(* CoDeSys 2.3 library: Lib_MQTT_Publisher_01.lib *)
(* Libraries: Lib_DebugLogger_01.lib 18.7.17 20:48:14, C:\Program Files (x86)\WAGO Software\CoDeSys V2.3\Targets\WAGO\Libraries\32_Bit\SysLibSockets.lib 10.2.11 09:20:54, C:\Program Files (x86)\WAGO Software\CoDeSys V2.3\Targets\WAGO\Libraries\Application\WagoLibEthernet_01.lib 1.4.15 14:24:28, Standard.lib 2.6.14 10:37:46, Util.lib 26.9.14 10:12:46 *)

(* Data type *)
TYPE Buffer :
STRUCT
	data : ARRAY [0..MAX_RECEIVE_TCP_CLIENT] OF BYTE;
	iPos : DWORD := 0;
END_STRUCT
END_TYPE

(* Data type *)
TYPE ConnectFlags :
STRUCT
	xUsername     : BOOL;
	xPassword     : BOOL;
	xWillRetain   : BOOL;
	xWillQoS1     : BOOL;
    xWillQoS2     : BOOL;
	xWillFlag     : BOOL;
	xCleanSession : BOOL;
END_STRUCT
END_TYPE

(* Data type *)
TYPE E_MQTT_MAIN_STATE : (

	eMQTT_NO_TCP_CONNECTION,
	eMQTT_CONNECTED,
	eMQTT_NOT_CONNECTED,
	eMQTT_TIMEOUT,
	eMQTT_WAIT_RESPONSE
);
END_TYPE

(* Data type *)
TYPE FixedHeader :
STRUCT
	bMessageType : BYTE := 16#00;
	xDUP_FLAG    : BOOL := FALSE;
	xQos         : BYTE := 16#00; (*0,1,2*)
	xRetain      : BOOL := FALSE;
END_STRUCT
END_TYPE

(* Data type *)
TYPE stMQTT_Config :
STRUCT
	sIdentifier : STRING := 'wagoPLC';
	sIp : STRING;
	wPortNumber : WORD := 1883;
	sUsername : STRING;
	sPassword : STRING;
END_STRUCT
END_TYPE

(* POU _BUFFER_CONCAT, ST *)
FUNCTION _BUFFER_CONCAT : BOOL
VAR_INPUT
	PT  : POINTER TO Buffer;
	PTContact  : POINTER TO Buffer;
END_VAR
VAR
	i: INT;
END_VAR
FOR i:=0 TO DWORD_TO_INT(PTContact^.iPos) -1 BY 1 DO
	_BUFFER_PUSH(PT, PTContact^.data[i]);
END_FOR
END_FUNCTION

(* POU _BUFFER_PUSH, ST *)
FUNCTION _BUFFER_PUSH : BOOL
VAR_INPUT
	PT  : POINTER TO Buffer;
	IN  : BYTE;
END_VAR

VAR
END_VAR
(* pushed data to a buffer array *)
PT^.data[PT^.iPos] := IN;

PT^.iPos := PT^.iPos + 1;

_BUFFER_PUSH := TRUE;
END_FUNCTION

(* POU _BUFFER_PUSH_STRING, ST *)
FUNCTION _BUFFER_PUSH_STRING : BOOL
VAR_INPUT
	PT : POINTER TO Buffer;
	IN : STRING(255);
	INCLUDE_LENGTH : BOOL := FALSE;
END_VAR
VAR
	sPT : POINTER TO BYTE;
	iLen : DWORD;
	i : DWORD;
	nxtPtr: POINTER TO BYTE;
END_VAR
iLen := LEN(IN);
sPT := ADR(IN);

IF INCLUDE_LENGTH THEN

(*
	_BUFFER_PUSH(PT, BYTE_OF_DWORD(iLen,1));
	_BUFFER_PUSH(PT, BYTE_OF_DWORD(iLen,0));
*)

		_BUFFER_PUSH(PT, DWORD_TO_BYTE(SHR(iLen,8)));
		_BUFFER_PUSH(PT, DWORD_TO_BYTE(iLen));

END_IF

FOR i:=0 TO iLen-1 BY 1 DO
	nxtPtr := sPT + i * SIZEOF(sPT^);
	_BUFFER_PUSH(PT, nxtPtr^);
END_FOR
END_FUNCTION

(* POU _BUFFER_SET, ST *)
FUNCTION _BUFFER_SET : BOOL
VAR_INPUT
	PT  : POINTER TO Buffer;
	IN  : BYTE;
	POS : UINT := 0;
END_VAR
VAR
END_VAR
PT^.data[POS] := IN;

IF PT^.iPos < POS THEN
	PT^.iPos := POS;
END_IF
END_FUNCTION

(* POU CREATE_MESSAGE, ST *)
FUNCTION CREATE_MESSAGE : BOOL
VAR_INPUT
	PT          : POINTER TO Buffer;
	fixedHeader     : FixedHeader;
	variableHeader  : Buffer;
	payLoad         : Buffer;
END_VAR
VAR
	bTemp  : BYTE;
	remainingLength: DWORD;
END_VAR
(* FIXED HEADER *)
(* BYTE 1 *)
bTemp := bTemp OR SHL(fixedHeader.bMessageType, 4) OR SHL(FixedHeader.xQos, 1);

bTemp.3 := FixedHeader.xDUP_FLAG;
bTemp.0 := FixedHeader.xRetain;

_BUFFER_PUSH(PT, bTemp);

(* BYTE 2 *)
remainingLength := variableHeader.iPos + payLoad.iPos;

ENCODE_REMAINING_LENGTH(PT, remainingLength);
(*_BUFFER_PUSH(PT, remainingLength);*)

(* VARIABLE HEADER *)
_BUFFER_CONCAT(PT, ADR(variableHeader));

(* PAYLOAD *)
_BUFFER_CONCAT(PT, ADR(payLoad));
END_FUNCTION

(* POU ENCODE_REMAINING_LENGTH, ST *)
FUNCTION ENCODE_REMAINING_LENGTH : BOOL
VAR_INPUT
	PT : POINTER TO Buffer;
	LENGTH : DWORD;
END_VAR
VAR
	wPt : POINTER TO DWORD; (*4 bytes*)
	digit: DWORD;
END_VAR
wPt := ADR(LENGTH);

IF LENGTH = 0 THEN
	_BUFFER_PUSH(PT, 16#00);
	RETURN;
END_IF

WHILE LENGTH > 0 DO
	digit := LENGTH MOD 128;
	LENGTH := LENGTH / 128;
	
	IF LENGTH > 0 THEN
		digit := digit OR 16#80;
	END_IF
(*	_BUFFER_PUSH(PT, BYTE_OF_DWORD(digit,0));*)
	_BUFFER_PUSH(PT, DWORD_TO_BYTE(digit));
END_WHILE
END_FUNCTION

(* POU MQTT_Client, ST *)
FUNCTION_BLOCK MQTT_Client

VAR_INPUT
	sTopic: STRING;
	sPayload: STRING(255);
	sIp : STRING;
	iPortNumber : WORD;
	sUsername : STRING;
	sPassword : STRING;
END_VAR

VAR_IN_OUT
	xPublish: BOOL;
END_VAR

VAR_OUTPUT
	xConnected : BOOL := FALSE;
	xBusy : BOOL := FALSE;
END_VAR

VAR
	sendBuffer : 				Buffer;
	receiveBuffer :				Buffer;

	fixedHeader: 				FixedHeader;
	variableHeader: 			Buffer;

	payLoad:  					Buffer;

	connectFlags: 			ConnectFlags;
	tcpClient: 					TCP_Client;
	xStartSend 					: BOOL 					:= FALSE;
	diReceiveCount 				: DINT;
	connectionTimer				: TON;
	xTimeOut 					: BOOL;
	iIncomingMessageType		: BYTE;
	eState						: E_MQTT_MAIN_STATE 	:= eMQTT_NO_TCP_CONNECTION;
	xStartTimer					: BOOL;


	xOpenConnection: BOOL;



	bEntry: BOOL := TRUE;
	DebugLog: BOOL;
END_VAR

VAR CONSTANT
	CONNECTION_TIMEOUT : TIME := t#10s;


	Reserved   	: BYTE := 0;
	CONNECT     : BYTE := 1;
	CONNACK     : BYTE := 2;
	PUBLISH     : BYTE := 3;
	PUBACK      : BYTE := 4;
	PUBREC      : BYTE := 5;
	PUBREL      : BYTE := 6;
	PUBCOMP     : BYTE := 7;
	SUBSCRIBE   : BYTE := 8;
	SUBACK      : BYTE := 9;
	UNSUBSCRIBE : BYTE := 10;
	UNSUBACK    : BYTE := 11;
	PINGREQ     : BYTE := 12;
	PINGRESP    : BYTE := 13;
	DISCONNECT  : BYTE := 14;
	Reserved2   : BYTE := 15;

END_VAR
tcpClient(
	xOpenConnection		:= xOpenConnection,
	sIPaddress			:= sIp ,
	wPortNumber			:= iPortNumber,
	ptSendData 			:= ADR(sendBuffer.data),
	diSendCount 			:= sendBuffer.iPos,
	xStartSend 			:= xStartSend,
	aReceiveBuffer		:= receiveBuffer.data,
	diReceiveCount		:= diReceiveCount ,
	xConnected=> ,
	diError=> );

connectionTimer(
	IN:=xStartTimer,
	PT:=CONNECTION_TIMEOUT-t#2s,
	Q => xTimeOut);

(* INIT *)
payLoad.iPos := 0;
variableHeader.iPos := 0;

IF xTimeOut THEN
	eState := eMQTT_TIMEOUT;
END_IF

(* Execute current state *)

(*Global TCP Connection Check*)

IF 		(NOT tcpClient.xConnected OR tcpClient.diError <> 0)
	AND eState <> eMQTT_NO_TCP_CONNECTION THEN
	DebugLog('connection lost', INFO);
	DebugLog(DINT_TO_STRING(tcpClient.diError), INFO);
	eState := eMQTT_NO_TCP_CONNECTION;
	bEntry := TRUE;
END_IF;



CASE eState OF


	eMQTT_NO_TCP_CONNECTION:
		IF bEntry THEN
			bEntry := FALSE;
			xOpenConnection := FALSE;
			xStartSend := FALSE;
			xConnected := FALSE;
			DebugLog('try to connect', INFO);

		ELSE
			xOpenConnection := TRUE;
			IF tcpClient.xConnected THEN
				eState := eMQTT_NOT_CONNECTED;
				bEntry := TRUE;
			END_IF

		END_IF




	eMQTT_CONNECTED:
			IF diReceiveCount > 0 THEN
				iIncomingMessageType := receiveBuffer.data[0];
				IF iIncomingMessageType = SHL(PINGRESP, 4) THEN
					xStartTimer := TRUE;
				END_IF
				diReceiveCount := 0;
			END_IF
	
			IF xPublish THEN
				fixedHeader.bMessageType := PUBLISH;
				fixedHeader.xDUP_FLAG := FALSE;
				fixedHeader.xQos := 16#00; (* only QoS 0 supported *)
				fixedHeader.xRetain := FALSE;
		
				_BUFFER_PUSH_STRING(ADR(variableHeader), sTopic, TRUE); (* Topic *)
				IF fixedHeader.xQos > 16#00 THEN
					_BUFFER_PUSH(ADR(variableHeader), 16#00);(* Message ID *)
					_BUFFER_PUSH(ADR(variableHeader), 16#00);
				END_IF
	
				_BUFFER_PUSH_STRING(ADR(payLoad), sPayload, FALSE);
		
				sendBuffer.iPos := 0;
				CREATE_MESSAGE(ADR(sendBuffer), fixedHeader, variableHeader, payLoad);
	
				xStartSend := TRUE;
		
				xPublish := FALSE;

			END_IF



	eMQTT_NOT_CONNECTED:

			sendBuffer.iPos := 0;
			xStartTimer := FALSE;
			fixedHeader.bMessageType := CONNECT;
	
			_BUFFER_PUSH_STRING(
				ADR(variableHeader),
				'MQIsdp',
				TRUE); (* Protocol Name*)
			_BUFFER_PUSH(
				ADR(variableHeader),
				 3); (* Version Number*)
	
			connectFlags.xCleanSession 	:= TRUE;
			connectFlags.xWillFlag     		:= FALSE;
			connectFlags.xWillQoS1    	 	:= FALSE;
			connectFlags.xWillQoS2     		:= FALSE;
			connectFlags.xWillRetain   		:= FALSE;
			connectFlags.xUsername 		:= LEN(sUsername) > 0;
			connectFlags.xPassword 		:= LEN(sPassword) > 0;
	
			_BUFFER_PUSH(
				ADR(variableHeader),
				 PACK(		FALSE,
							connectFlags.xCleanSession,
							connectFlags.xWillFlag,
							connectFlags.xWillQoS1,
							connectFlags.xWillQoS2,
							connectFlags.xWillRetain,
							connectFlags.xPassword,
							connectFlags.xUsername));
	
			_BUFFER_PUSH(ADR(variableHeader), 16#00);
			_BUFFER_PUSH(ADR(variableHeader), 16#0A); (* Keep Alive: 10s *)
			_BUFFER_PUSH_STRING(ADR(payload), 'PLC', TRUE); (* Client Identfier *)
	
			IF connectFlags.xUsername THEN
				_BUFFER_PUSH_STRING(ADR(payload), sUsername, TRUE); (* Username *)
			END_IF
	
			IF connectFlags.xPassword THEN
				_BUFFER_PUSH_STRING(ADR(payload), sPassword, TRUE); (* Password *)
			END_IF
	
			CREATE_MESSAGE(ADR(sendBuffer), fixedHeader, variableHeader, payLoad);

			xStartSend := TRUE;
			bEntry := TRUE;
			eState := eMQTT_WAIT_RESPONSE;



	eMQTT_TIMEOUT:


		sendBuffer.iPos := 0;
		xStartTimer := FALSE	;
		fixedHeader.bMessageType := PINGREQ;
		CREATE_MESSAGE(ADR(sendBuffer), fixedHeader, variableHeader, payLoad);
	
		eState :=eMQTT_CONNECTED;
		xStartSend := TRUE;


	eMQTT_WAIT_RESPONSE:
		iIncomingMessageType := receiveBuffer.data[0];
		IF iIncomingMessageType = SHL(CONNACK, 4) THEN
			(* TODO: Check return code *)
			xConnected := TRUE;
			xStartTimer := TRUE;
			bEntry := TRUE;
			eState := eMQTT_CONNECTED;
			diReceiveCount := 0;
		END_IF

END_CASE


xBusy := xStartSend;
END_FUNCTION_BLOCK

(* Visualisation PLC_VISU
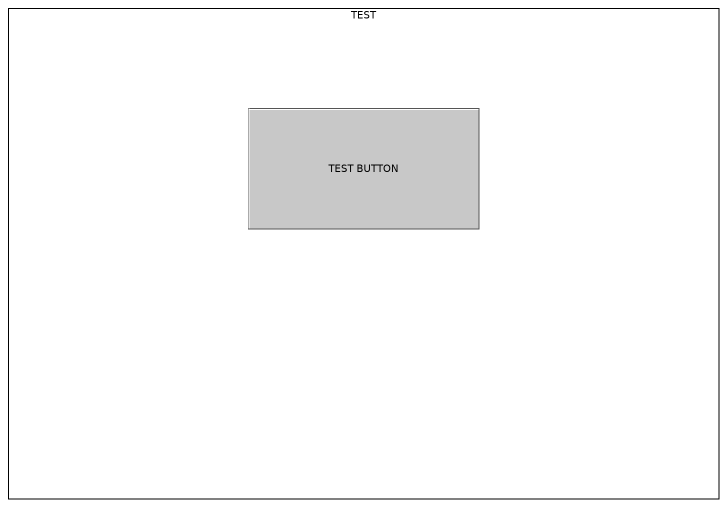
rectangle at (30,10)-(741,501): text "TEST"
button at (270,110)-(501,231): text "TEST BUTTON"
*)
